PROGRAM MAIN
VAR
	fFahrenheit : REAL;
END_VAR

fFahrenheit := Celsius_To_Fahrenheit(fCelsius := 5.0);

END_PROGRAM

(* stored: Version 1.1.0.1, ProductVersion 3.1.4024.11
   POU MAIN: Id {dff884c8-a5df-44c5-b67a-7ce68b89575f}, SpecialFunc None *)
